{attribute addProperty BoxType "EJ4132-0000-0019"}
{attribute addProperty Id "AO_Outputs_ChannelAT %Q*ARRAY[0..1] OF AO_Outputs_Channel_F57FA4F93240WcStateAT %I*WcState_64F6A8C6810InfoDataAT %I*InfoData_BC63D37F80100"}
{attribute addProperty CRC "2182094866"}
{attribute addProperty SizeInBites "120"}
{attribute addProperty SizeInBytes "15"}
TYPE EJ4132_08E1E1D8 :
STRUCT
	{attribute addProperty Name "AO_Outputs_Channel"}
	AO_Outputs_Channel : ARRAY[0..1] OF AO_Outputs_Channel_F57FA4F9;
	{attribute addProperty Name "WcState"}
	WcState : WcState_64F6A8C6;
	{attribute addProperty Name "InfoData"}
	InfoData : InfoData_BC63D37F;
END_STRUCT
END_TYPE

(* stored: Version 1.2.0.0, ProductVersion 3.1.4024.9
   DUT EJ4132_08E1E1D8: Id {715d30ab-adff-424e-9575-2b0a8a18cc89} *)
